(* Logix 5000 project; controller VET 1756-L62 rev 19.52; software revision 19.01; part 16 of 27 *)
(* tags used below, declared in another part *)
   _Eqp : Equipo[800];
   Batch : batch[10];
   dosificador : dosif_struct[20];
   Dosificar_MIC_02 : PHASE;
   Dosificar_MID_01 : PHASE;
   fecha_plc : DINT;
   hora_plc : DINT;
   SetDInt : DINT[500];
   TabBin : Bins_Setup;
   Timer : TIMER[500];
   vdf : VDFS[20];
(* Dosificar_MIC_02, continued *)

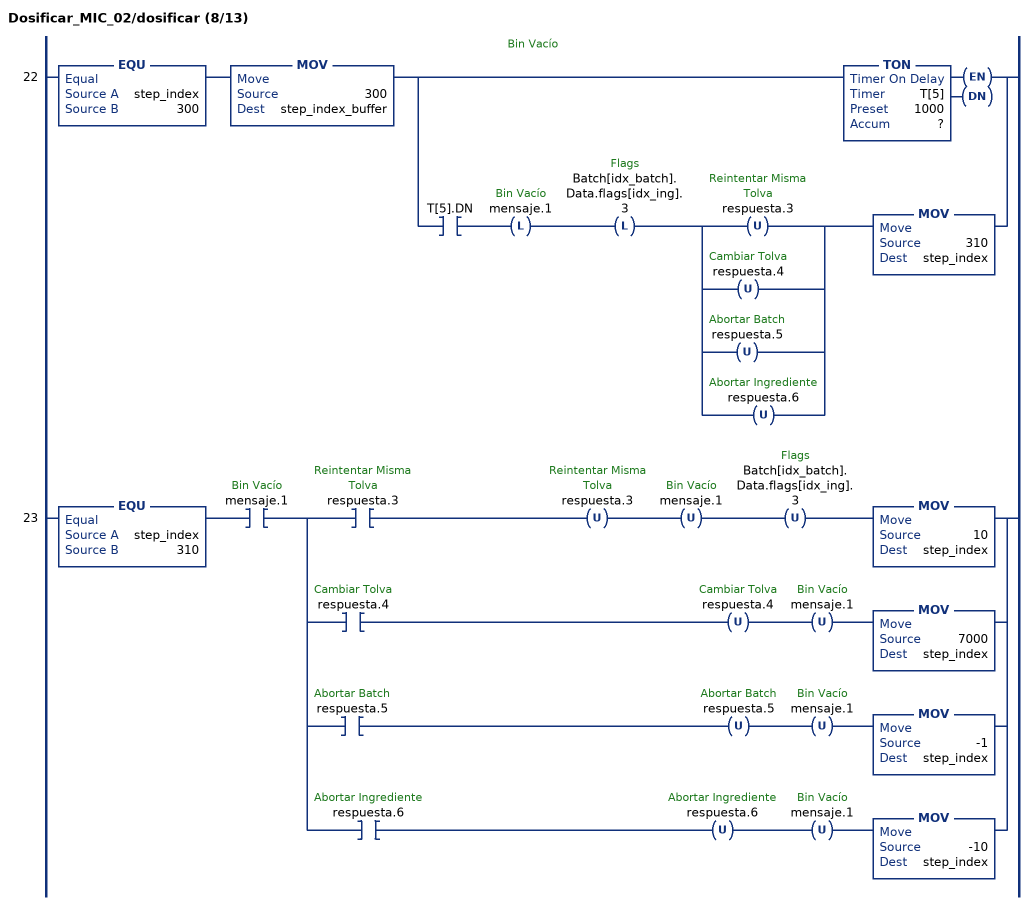
   // Bin Vacío
   22: EQU(step_index,300)MOV(300,step_index_buffer)[TON(T[5],?,?) ,XIC(T[5].DN) OTL(mensaje.1) OTL(Batch[idx_batch].Data.flags[idx_ing].3) [OTU(respuesta.3) ,OTU(respuesta.4) ,OTU(respuesta.5) ,OTU(respuesta.6) ] MOV(310,step_index) ];
   23: EQU(step_index,310)XIC(mensaje.1)[XIC(respuesta.3) OTU(respuesta.3) OTU(mensaje.1) OTU(Batch[idx_batch].Data.flags[idx_ing].3) MOV(10,step_index) ,XIC(respuesta.4) OTU(respuesta.4) OTU(mensaje.1) MOV(7000,step_index) ,XIC(respuesta.5) OTU(respuesta.5) OTU(mensaje.1) MOV(-1,step_index) ,XIC(respuesta.6) OTU(respuesta.6) OTU(mensaje.1) MOV(-10,step_index) ];
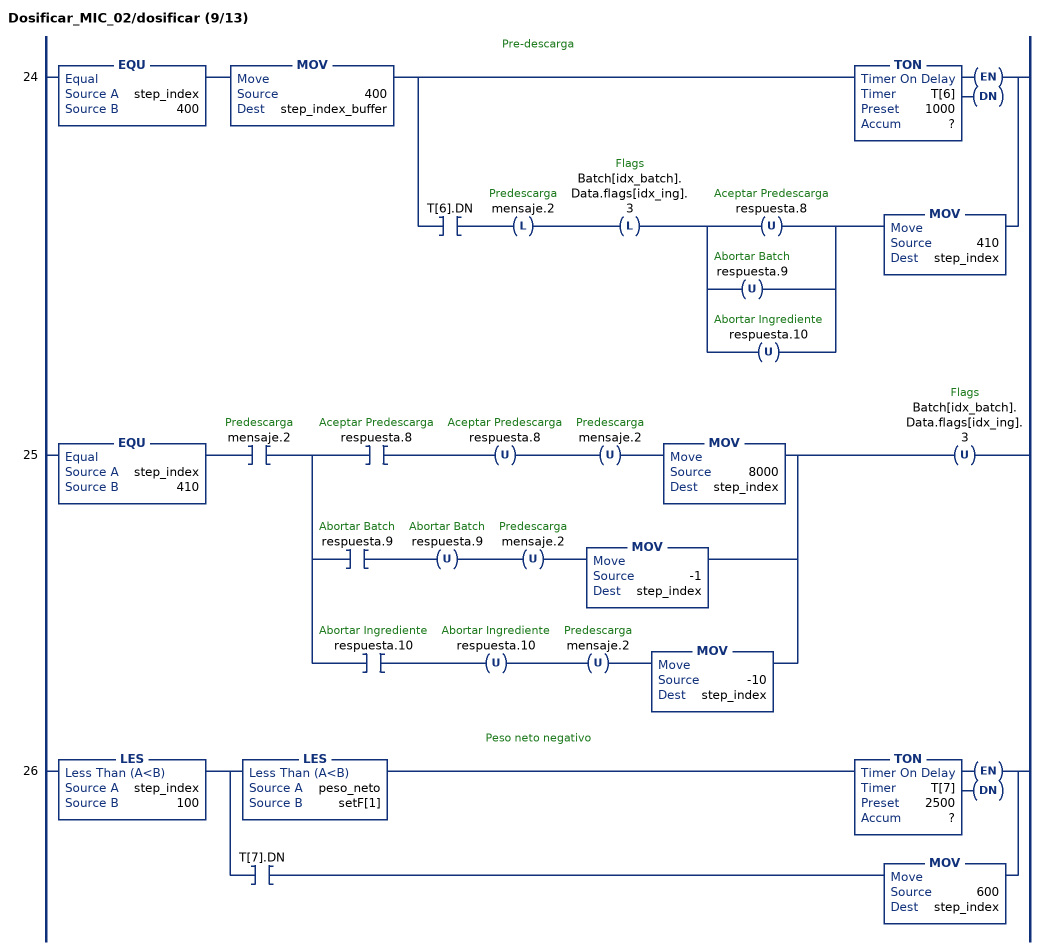
   // Pre-descarga
   24: EQU(step_index,400)MOV(400,step_index_buffer)[TON(T[6],?,?) ,XIC(T[6].DN) OTL(mensaje.2) OTL(Batch[idx_batch].Data.flags[idx_ing].3) [OTU(respuesta.8) ,OTU(respuesta.9) ,OTU(respuesta.10) ] MOV(410,step_index) ];
   25: EQU(step_index,410)XIC(mensaje.2)[XIC(respuesta.8) OTU(respuesta.8) OTU(mensaje.2) MOV(8000,step_index) ,XIC(respuesta.9) OTU(respuesta.9) OTU(mensaje.2) MOV(-1,step_index) ,XIC(respuesta.10) OTU(respuesta.10) OTU(mensaje.2) MOV(-10,step_index) ]OTU(Batch[idx_batch].Data.flags[idx_ing].3);
   // Peso neto negativo
   26: LES(step_index,100)[LES(peso_neto,setF[1]) TON(T[7],?,?) ,XIC(T[7].DN) MOV(600,step_index) ];
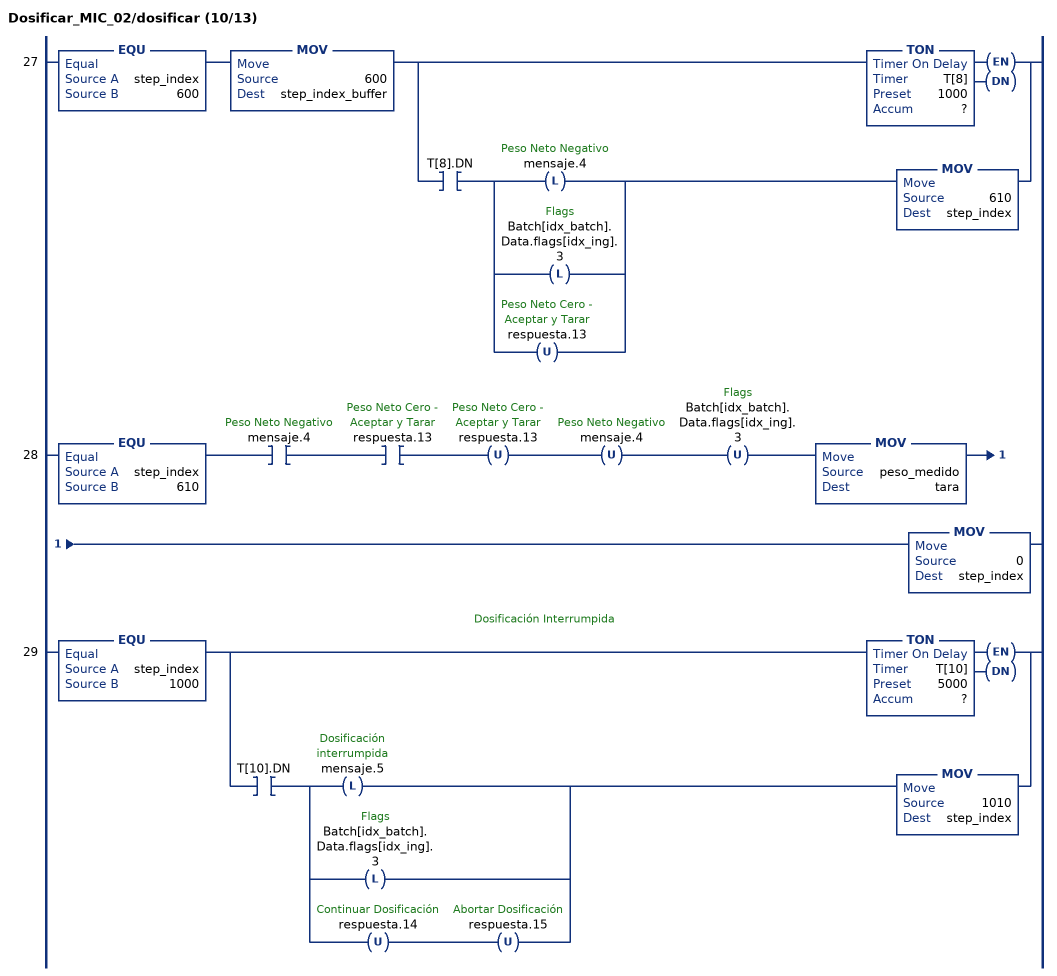
   27: EQU(step_index,600)MOV(600,step_index_buffer)[TON(T[8],?,?) ,XIC(T[8].DN) [OTL(mensaje.4) ,OTL(Batch[idx_batch].Data.flags[idx_ing].3) ,OTU(respuesta.13) ] MOV(610,step_index) ];
   28: EQU(step_index,610)XIC(mensaje.4)XIC(respuesta.13)OTU(respuesta.13)OTU(mensaje.4)OTU(Batch[idx_batch].Data.flags[idx_ing].3)MOV(peso_medido,tara)MOV(0,step_index);
   // Dosificación Interrumpida
   29: EQU(step_index,1000)[TON(T[10],?,?) ,XIC(T[10].DN) [OTL(mensaje.5) ,OTL(Batch[idx_batch].Data.flags[idx_ing].3) ,OTU(respuesta.14) OTU(respuesta.15) ] MOV(1010,step_index) ];
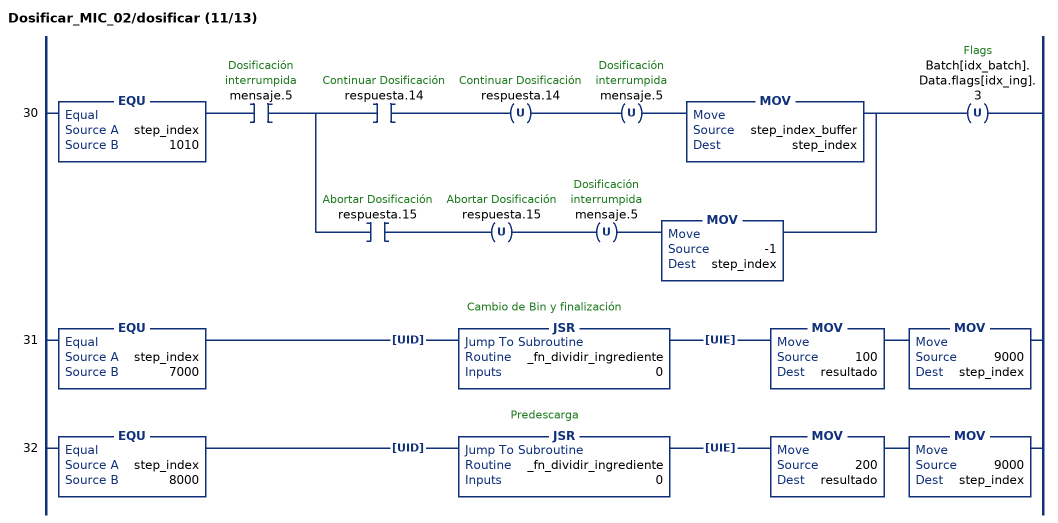
   30: EQU(step_index,1010)XIC(mensaje.5)[XIC(respuesta.14) OTU(respuesta.14) OTU(mensaje.5) MOV(step_index_buffer,step_index) ,XIC(respuesta.15) OTU(respuesta.15) OTU(mensaje.5) MOV(-1,step_index) ]OTU(Batch[idx_batch].Data.flags[idx_ing].3);
   // Cambio de Bin y finalización
   31: EQU(step_index,7000)UID()JSR(_fn_dividir_ingrediente,0)UIE()MOV(100,resultado)MOV(9000,step_index);
   // Predescarga
   32: EQU(step_index,8000)UID()JSR(_fn_dividir_ingrediente,0)UIE()MOV(200,resultado)MOV(9000,step_index);
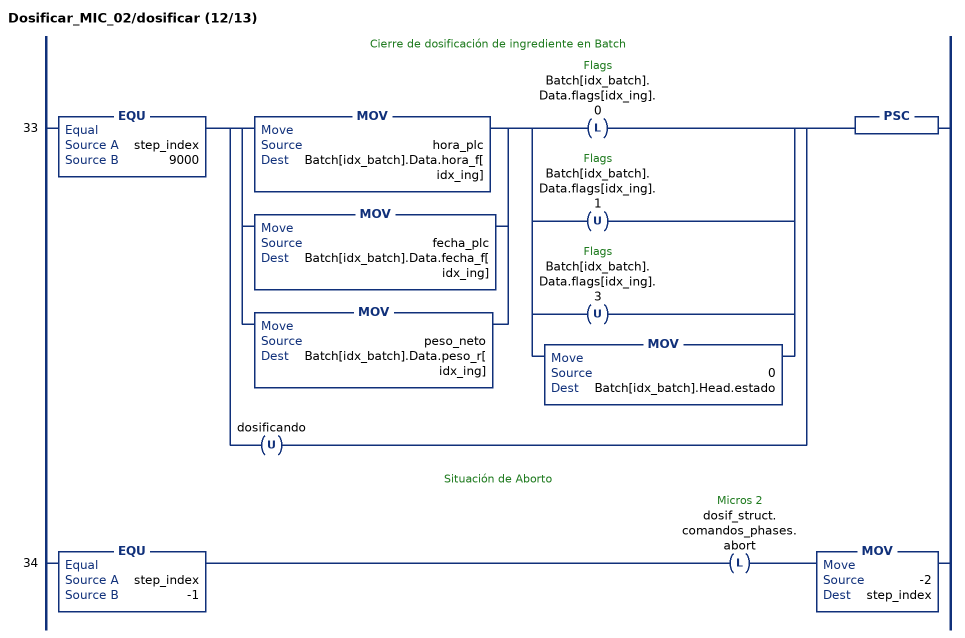
   // Cierre de dosificación de ingrediente en Batch
   33: EQU(step_index,9000)[[MOV(hora_plc,Batch[idx_batch].Data.hora_f[idx_ing]) ,MOV(fecha_plc,Batch[idx_batch].Data.fecha_f[idx_ing]) ,MOV(peso_neto,Batch[idx_batch].Data.peso_r[idx_ing]) ] [OTL(Batch[idx_batch].Data.flags[idx_ing].0) ,OTU(Batch[idx_batch].Data.flags[idx_ing].1) ,OTU(Batch[idx_batch].Data.flags[idx_ing].3) ,MOV(0,Batch[idx_batch].Head.estado) ] ,OTU(dosificando) ]PSC();
   // Situación de Aborto
   34: EQU(step_index,-1)OTL(dosif_struct.comandos_phases.abort)MOV(-2,step_index);
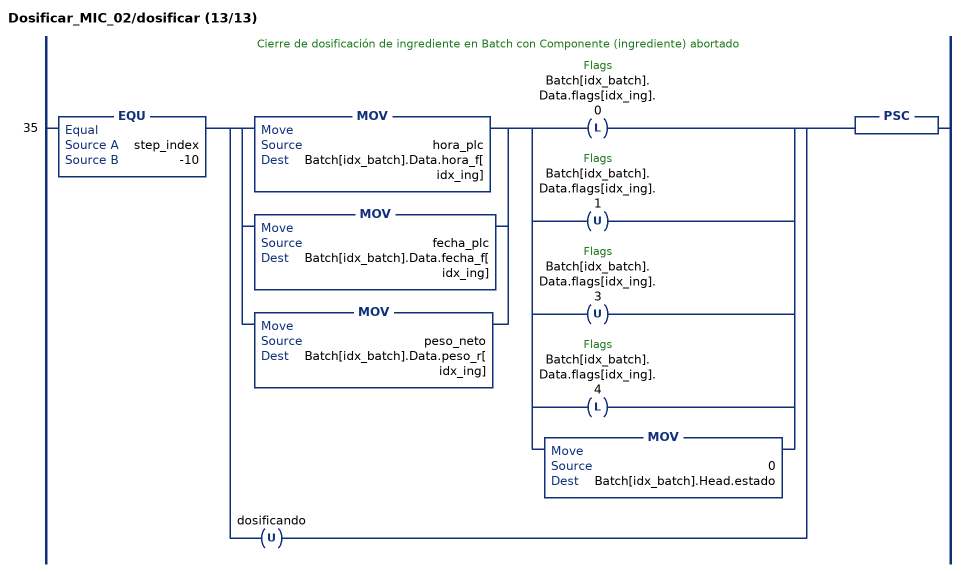
   // Cierre de dosificación de ingrediente en Batch con Componente (ingrediente) abortado
   35: EQU(step_index,-10)[[MOV(hora_plc,Batch[idx_batch].Data.hora_f[idx_ing]) ,MOV(fecha_plc,Batch[idx_batch].Data.fecha_f[idx_ing]) ,MOV(peso_neto,Batch[idx_batch].Data.peso_r[idx_ing]) ] [OTL(Batch[idx_batch].Data.flags[idx_ing].0) ,OTU(Batch[idx_batch].Data.flags[idx_ing].1) ,OTU(Batch[idx_batch].Data.flags[idx_ing].3) ,OTL(Batch[idx_batch].Data.flags[idx_ing].4) ,MOV(0,Batch[idx_batch].Head.estado) ] ,OTU(dosificando) ]PSC();
END_ROUTINE

ROUTINE Falla   (* ladder *)
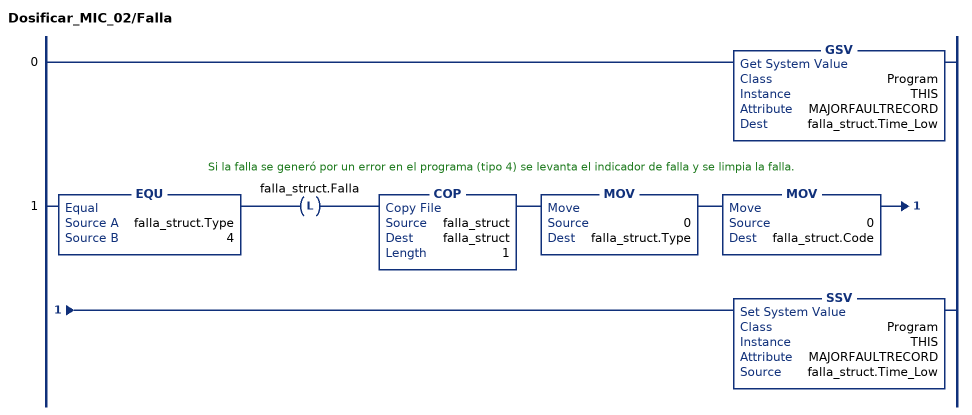
   0: GSV(Program,THIS,MAJORFAULTRECORD,falla_struct.Time_Low);
   // Si la falla se generó por un error en el programa (tipo 4) se levanta el indicador de falla y se limpia la falla.
   1: EQU(falla_struct.Type,4)OTL(falla_struct.Falla)COP(falla_struct,falla_struct,1)MOV(0,falla_struct.Type)MOV(0,falla_struct.Code)SSV(Program,THIS,MAJORFAULTRECORD,falla_struct.Time_Low);
END_ROUTINE

ROUTINE Holding   (* ladder *)
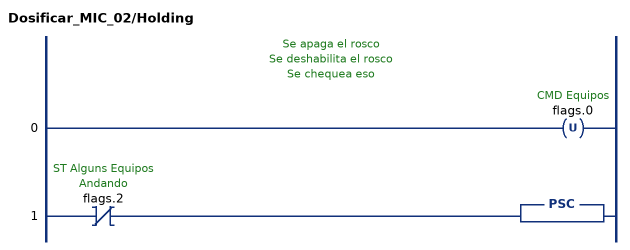
   // Se apaga el rosco
   // Se deshabilita el rosco
   // Se chequea eso
   0: OTU(flags.0);
   1: XIO(flags.2)PSC();
END_ROUTINE

ROUTINE preState   (* ladder *)
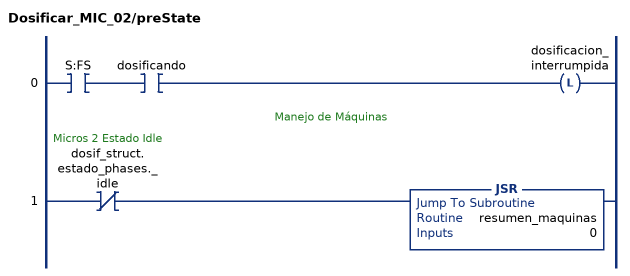
   0: XIC(S:FS)XIC(dosificando)OTL(dosificacion_interrumpida);
   // Manejo de Máquinas
   1: XIO(dosif_struct.estado_phases._idle)JSR(resumen_maquinas,0);
END_ROUTINE

ROUTINE Resetting   (* ladder *)
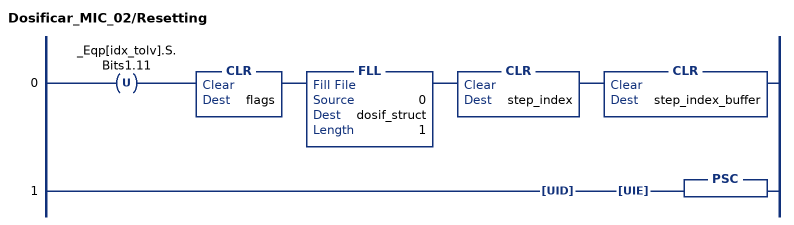
   0: OTU(_Eqp[idx_tolv].S.Bits1.11)CLR(flags)FLL(0,dosif_struct,1)CLR(step_index)CLR(step_index_buffer);
   1: UID()UIE()PSC();
END_ROUTINE

ROUTINE Restarting   (* ladder *)
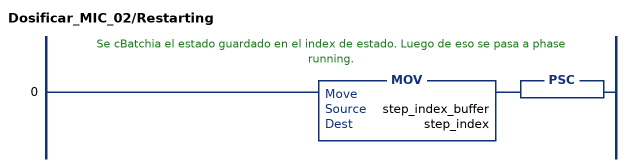
   // Se cBatchia el estado guardado en el index de estado. Luego de eso se pasa a phase running.
   0: MOV(step_index_buffer,step_index)PSC();
END_ROUTINE

ROUTINE resumen_maquinas   (* ladder *)
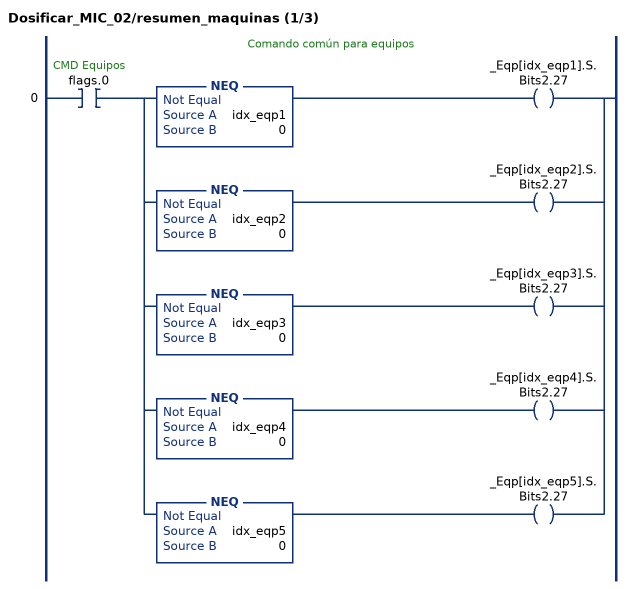
   // Comando común para equipos
   0: XIC(flags.0)[NEQ(idx_eqp1,0) OTE(_Eqp[idx_eqp1].S.Bits2.27) ,NEQ(idx_eqp2,0) OTE(_Eqp[idx_eqp2].S.Bits2.27) ,NEQ(idx_eqp3,0) OTE(_Eqp[idx_eqp3].S.Bits2.27) ,NEQ(idx_eqp4,0) OTE(_Eqp[idx_eqp4].S.Bits2.27) ,NEQ(idx_eqp5,0) OTE(_Eqp[idx_eqp5].S.Bits2.27) ];
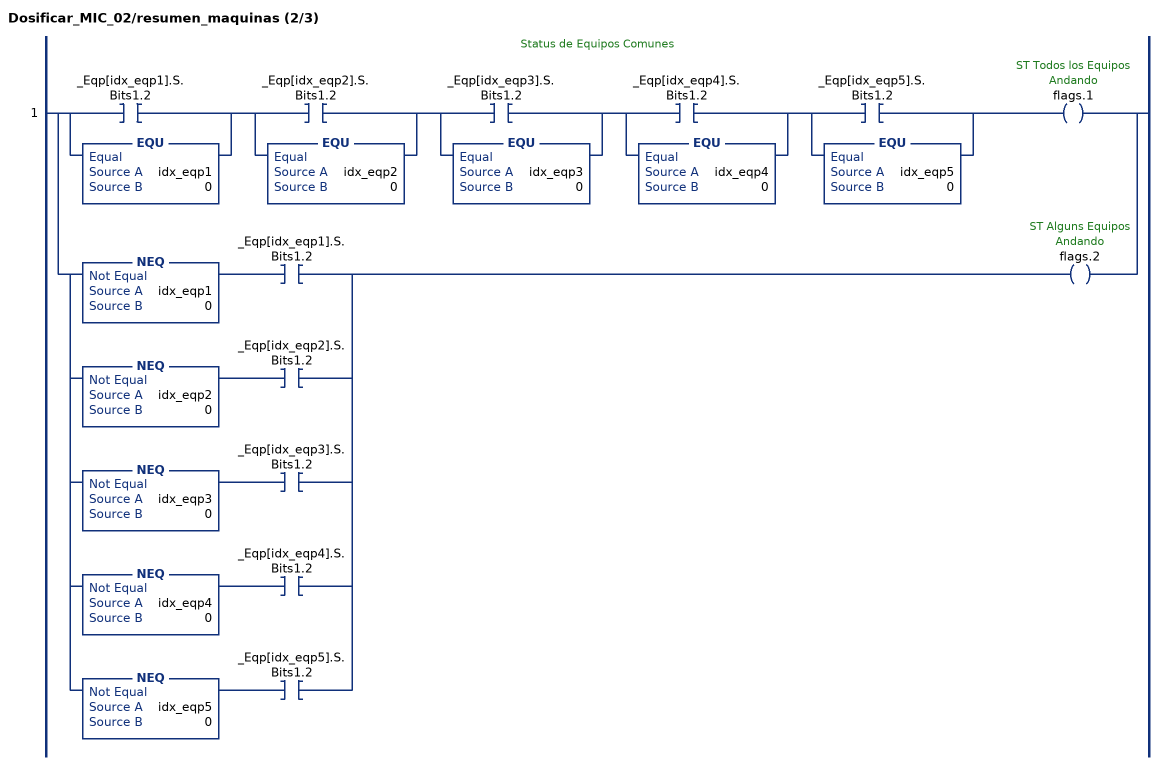
   // Status de Equipos Comunes
   1: [[XIC(_Eqp[idx_eqp1].S.Bits1.2) ,EQU(idx_eqp1,0) ] [XIC(_Eqp[idx_eqp2].S.Bits1.2) ,EQU(idx_eqp2,0) ] [XIC(_Eqp[idx_eqp3].S.Bits1.2) ,EQU(idx_eqp3,0) ] [XIC(_Eqp[idx_eqp4].S.Bits1.2) ,EQU(idx_eqp4,0) ] [XIC(_Eqp[idx_eqp5].S.Bits1.2) ,EQU(idx_eqp5,0) ] OTE(flags.1) ,[NEQ(idx_eqp1,0) XIC(_Eqp[idx_eqp1].S.Bits1.2) ,NEQ(idx_eqp2,0) XIC(_Eqp[idx_eqp2].S.Bits1.2) ,NEQ(idx_eqp3,0) XIC(_Eqp[idx_eqp3].S.Bits1.2) ,NEQ(idx_eqp4,0) XIC(_Eqp[idx_eqp4].S.Bits1.2) ,NEQ(idx_eqp5,0) XIC(_Eqp[idx_eqp5].S.Bits1.2) ] OTE(flags.2) ];
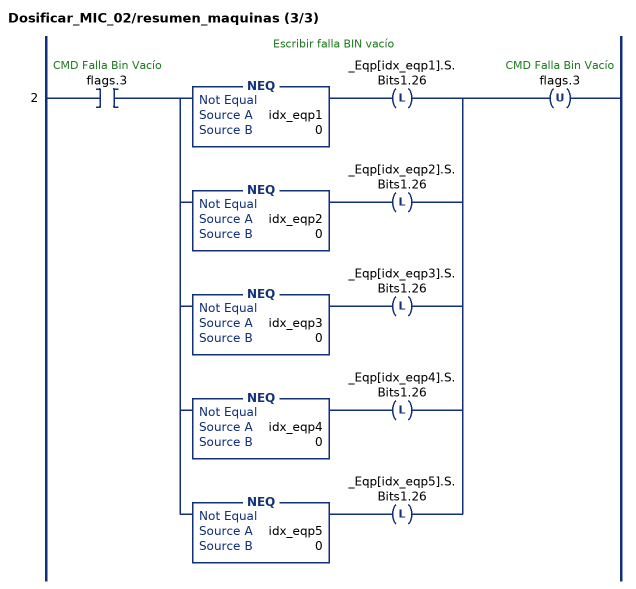
   // Escribir falla BIN vacío
   2: XIC(flags.3)[NEQ(idx_eqp1,0) OTL(_Eqp[idx_eqp1].S.Bits1.26) ,NEQ(idx_eqp2,0) OTL(_Eqp[idx_eqp2].S.Bits1.26) ,NEQ(idx_eqp3,0) OTL(_Eqp[idx_eqp3].S.Bits1.26) ,NEQ(idx_eqp4,0) OTL(_Eqp[idx_eqp4].S.Bits1.26) ,NEQ(idx_eqp5,0) OTL(_Eqp[idx_eqp5].S.Bits1.26) ]OTU(flags.3);
END_ROUTINE

ROUTINE Running   (* ladder *)
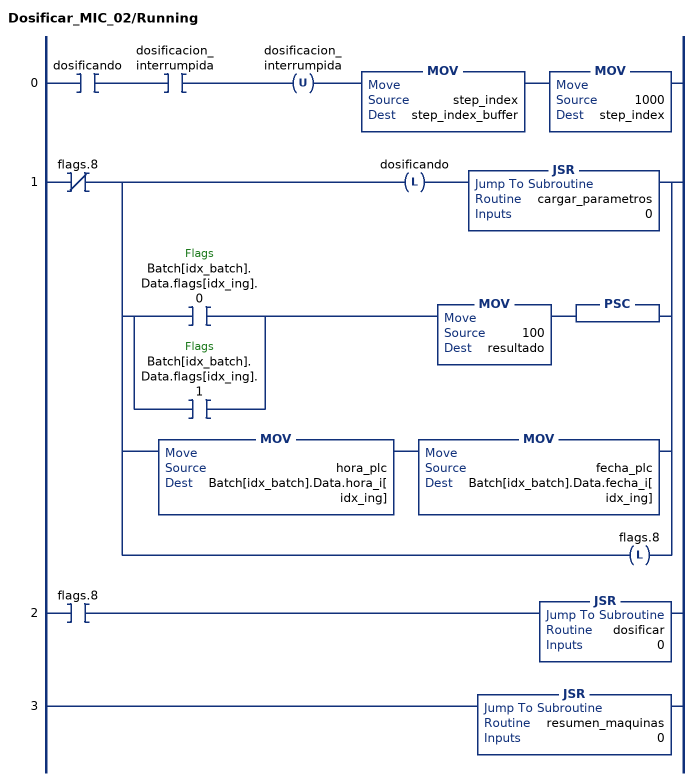
   0: XIC(dosificando)XIC(dosificacion_interrumpida)OTU(dosificacion_interrumpida)MOV(step_index,step_index_buffer)MOV(1000,step_index);
   1: XIO(flags.8)[OTL(dosificando) JSR(cargar_parametros,0) ,[[XIC(Batch[idx_batch].Data.flags[idx_ing].0) ,XIC(Batch[idx_batch].Data.flags[idx_ing].1) ] MOV(100,resultado) PSC() ,MOV(hora_plc,Batch[idx_batch].Data.hora_i[idx_ing]) MOV(fecha_plc,Batch[idx_batch].Data.fecha_i[idx_ing]) ] ,OTL(flags.8) ];
   2: XIC(flags.8)JSR(dosificar,0);
   3: JSR(resumen_maquinas,0);
END_ROUTINE
END_PROGRAM

PROGRAM Dosificar_MID_01   (* fault routine Falla *)
VAR
   _vel_exp : velocidad_exp := (x := 0.011880493, curvatura := 3.0, V_inicial := 70.0, V_final := 50.0, V_salida := 50.73287);
   bufferF : REAL[5] := ([0] := 90.78711, [1] := -0.7871094, [2] := 0.011880493);
        [2]   // Diferencia entre peso actual y objetivo
   debug : BOOL;
   dosif_extra_ingr : DINT := -1;   // Código del ingrediente que puede ser dosificado extra.
   dosif_struct : ALIAS FOR dosificador[1];
   dosificacion_interrumpida : BOOL;
   dosificando : BOOL;
   error_kg : REAL := 0.5;
   error_per : REAL := 4.5;
   falla_struct : falla_aux;
   flags : DINT;
        .1   // ST Todos los Equipos Andando
        .2   // ST Alguns Equipos Andando
        .3   // CMD Falla Bin Vacío
        .6   // Bit Precorte
        .7   // Aplicar Precorte
        .0   // CMD Equipos
   frq : ALIAS FOR dosif_struct.frq_terreno;
   frq_calculada : REAL := 50.0;
   frq_final : REAL := 50.0;
   frq_inicial : REAL := 70.0;
   hist_precorte : REAL[10] := ([0] := 1.0, [1] := 1.0, [2] := 1.0, [3] := 1.0, [4] := 1.0);
   i_fn : DINT;
   idx_batch : DINT := 3;
   idx_bin : DINT := 15;
   idx_dosif : DINT;   // Índice de dosificador usado
   idx_eqp1 : DINT := 53;
   idx_eqp2 : DINT;
   idx_eqp3 : DINT;
   idx_eqp4 : DINT;
   idx_eqp5 : DINT;
   idx_ing : DINT := 7;
   idx_tabbin : DINT := 1;
   idx_tolv : DINT := 34;   // Índice de Tolva
   limite_err_inf : REAL := 89.5;
   limite_err_sup : REAL := 90.5;
   mensaje : ALIAS FOR dosif_struct.msg;
        .1   // Bin Vacío
        .4   // Peso Neto Negativo
        .0   // Error de Pesaje
        .5   // Dosificación interrumpida
        .3   // Manual
        .2   // Predescarga
   peso_delta : REAL;
   peso_detencion : REAL := 89.09469;
   peso_intermedio : REAL := 54.000004;   // Peso límite para dosificación a frecuencia máxima
   peso_max : REAL := 700.0;
   peso_medido : ALIAS FOR dosif_struct.peso_terreno;
   peso_neto : REAL := 90.78711;
   peso_neto_aux : REAL;   // Peso Neto Guardado en caso de Vaciado y llenado de tolva
   peso_objetivo : REAL := 90.0;
   precorte : REAL := 1.102089;
   respuesta : ALIAS FOR dosif_struct.ans;
        .16   // Abortar Ingrediente
        .3   // Reintentar Misma Tolva
        .7   // Pasar a Manual
        .0   // Aceptar Error
        .14   // Continuar Dosificación
        .11   // Dosificación Completa
        .1   // Abortar Batch
        .2   // Abortar Ingrediente
        .12   // Habilitar Aceptar
        .8   // Aceptar Predescarga
        .10   // Abortar Ingrediente
        .5   // Abortar Batch
        .4   // Cambiar Tolva
        .6   // Abortar Ingrediente
        .15   // Abortar Dosificación
        .9   // Abortar Batch
        .13   // Peso Neto Cero - Aceptar y Tarar
   resultado : ALIAS FOR dosif_struct.resultado;
   return_fn : DINT;
   setD : DINT[5] := ([0] := 1, [1] := 44, [2] := 2, [3] := 1, [4] := 32);
        [1].3   // Aplicar Precorte
        [1].8   // Con VDF
        [4]   // Destino
        [1].2   // Predescarga
        [1].4   // Con Bloqueo de Tolva
        [1].5   // No respeta receta
        [2]   // Mezcladora izquierda
        [3]   // Mezcladora derecha
        [1].0   // Tipo LIW
        [0]   // Mínima variación de peso para detección de tolva vacía.
   setF : REAL[5] := ([0] := 1.0);
        [0]   // Límite para variación de peso
        [1]   // Límite para peso negativo
   step_index : DINT;
   step_index_buffer : DINT;
   T : TIMER[15] := ([0].PRE := 1000, [0].ACC := 80, [0].EN := 1, [0].TT := 1, [1].PRE := 30000, [2].PRE := 3000, [3].PRE := 10000, [4].PRE := 1000, [5].PRE := 1000, [6].PRE := 1000, [7].PRE := 2500, [8].PRE := 1000, [9].PRE := 1000, [10].PRE := 5000);
   t_espera : DINT := 3000;
   t_pulso : DINT := 10000;
   tara : REAL := 360.85922;
END_VAR

ROUTINE _fn_dividir_ingrediente   (* ladder *)
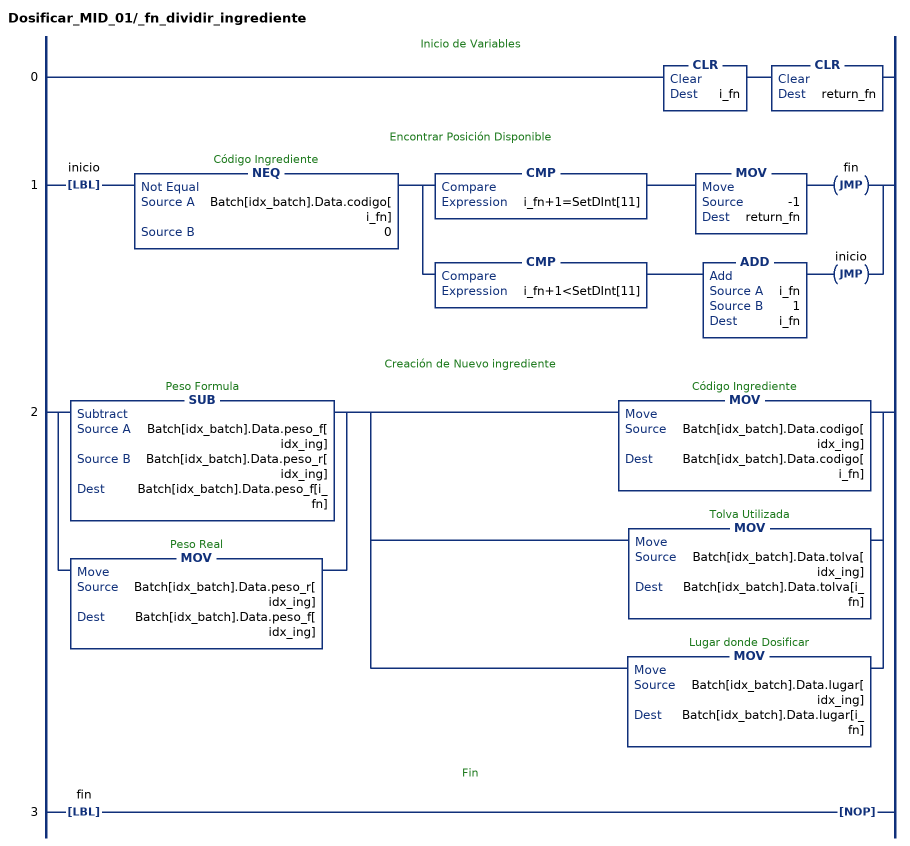
   // Inicio de Variables
   0: CLR(i_fn)CLR(return_fn);
   // Encontrar Posición Disponible
   1: LBL(inicio)NEQ(Batch[idx_batch].Data.codigo[i_fn],0)[CMP(i_fn+1=SetDInt[11]) MOV(-1,return_fn) JMP(fin) ,CMP(i_fn+1<SetDInt[11]) ADD(i_fn,1,i_fn) JMP(inicio) ];
   // Creación de Nuevo ingrediente
   2: [SUB(Batch[idx_batch].Data.peso_f[idx_ing],Batch[idx_batch].Data.peso_r[idx_ing],Batch[idx_batch].Data.peso_f[i_fn]) ,MOV(Batch[idx_batch].Data.peso_r[idx_ing],Batch[idx_batch].Data.peso_f[idx_ing]) ][MOV(Batch[idx_batch].Data.codigo[idx_ing],Batch[idx_batch].Data.codigo[i_fn]) ,MOV(Batch[idx_batch].Data.tolva[idx_ing],Batch[idx_batch].Data.tolva[i_fn]) ,MOV(Batch[idx_batch].Data.lugar[idx_ing],Batch[idx_batch].Data.lugar[i_fn]) ];
   // Fin
   3: LBL(fin)NOP();
END_ROUTINE

ROUTINE Aborting   (* ladder *)
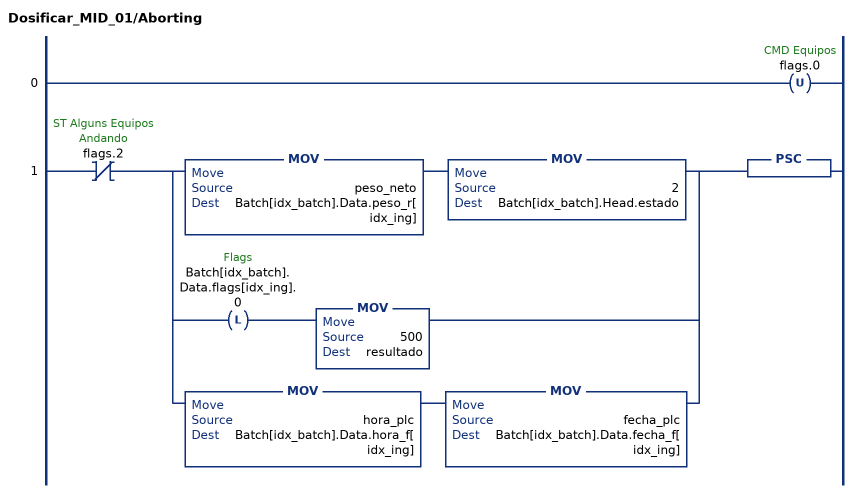
   0: OTU(flags.0);
   1: XIO(flags.2)[MOV(peso_neto,Batch[idx_batch].Data.peso_r[idx_ing]) MOV(2,Batch[idx_batch].Head.estado) ,OTL(Batch[idx_batch].Data.flags[idx_ing].0) MOV(500,resultado) ,MOV(hora_plc,Batch[idx_batch].Data.hora_f[idx_ing]) MOV(fecha_plc,Batch[idx_batch].Data.fecha_f[idx_ing]) ]PSC();
END_ROUTINE

ROUTINE calculo_frecuencia   (* ladder *)
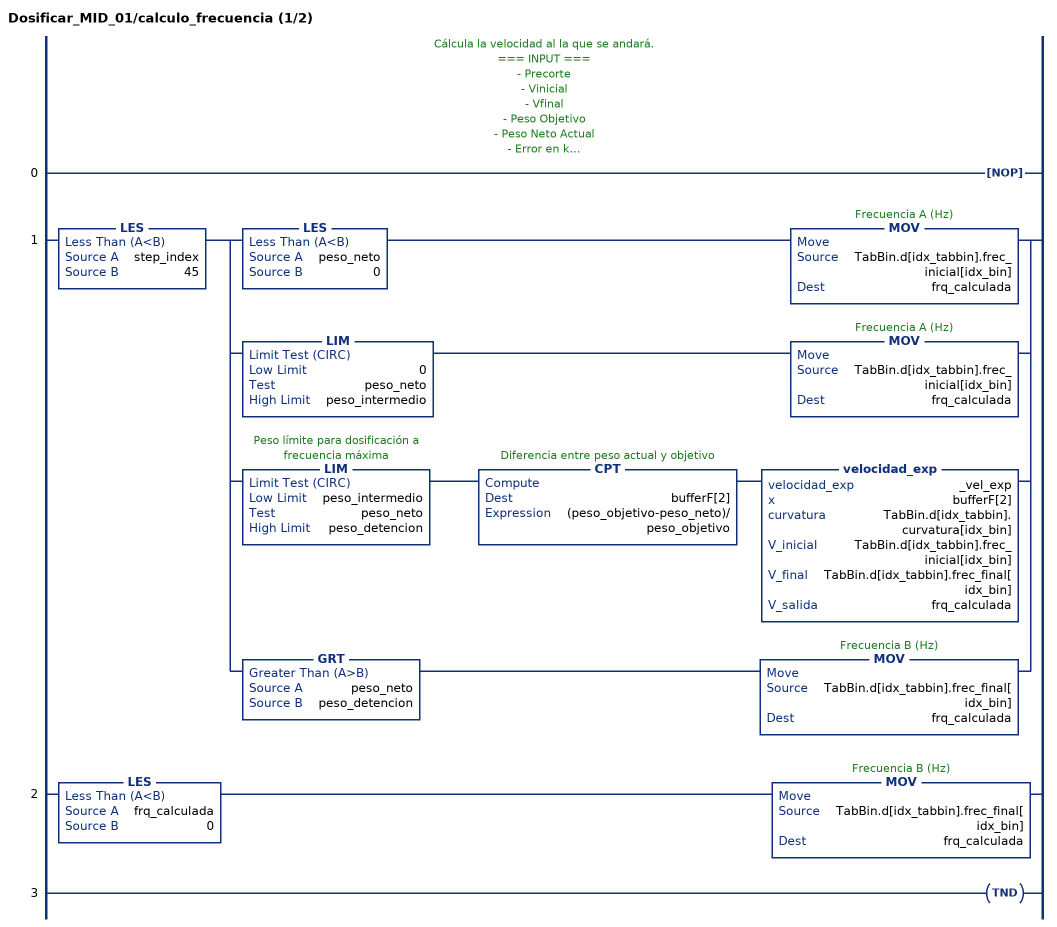
   // Cálcula la velocidad al la que se andará.
   // === INPUT ===
   // - Precorte
   // - Vinicial
   // - Vfinal
   // - Peso Objetivo
   // - Peso Neto Actual
   // - Error en kg
   // === OUTPUT ===
   // - Vactual
   0: NOP();
   1: LES(step_index,45)[LES(peso_neto,0) MOV(TabBin.d[idx_tabbin].frec_inicial[idx_bin],frq_calculada) ,LIM(0,peso_neto,peso_intermedio) MOV(TabBin.d[idx_tabbin].frec_inicial[idx_bin],frq_calculada) ,LIM(peso_intermedio,peso_neto,peso_detencion) CPT(bufferF[2],(peso_objetivo-peso_neto)/peso_objetivo) velocidad_exp(_vel_exp,bufferF[2],TabBin.d[idx_tabbin].curvatura[idx_bin],TabBin.d[idx_tabbin].frec_inicial[idx_bin],TabBin.d[idx_tabbin].frec_final[idx_bin],frq_calculada) ,GRT(peso_neto,peso_detencion) MOV(TabBin.d[idx_tabbin].frec_final[idx_bin],frq_calculada) ];
   2: LES(frq_calculada,0)MOV(TabBin.d[idx_tabbin].frec_final[idx_bin],frq_calculada);
   3: TND();
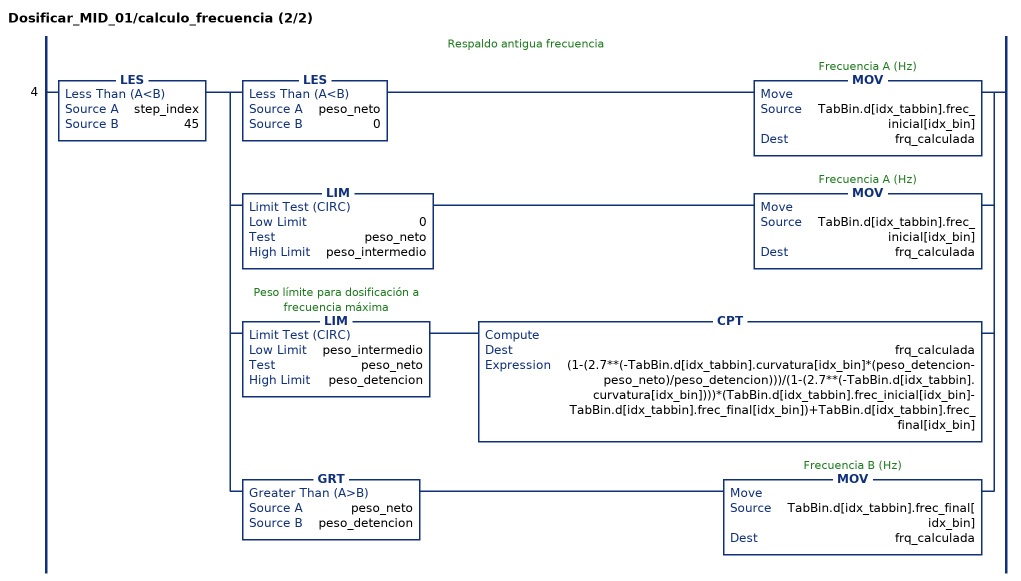
   // Respaldo antigua frecuencia
   4: LES(step_index,45)[LES(peso_neto,0) MOV(TabBin.d[idx_tabbin].frec_inicial[idx_bin],frq_calculada) ,LIM(0,peso_neto,peso_intermedio) MOV(TabBin.d[idx_tabbin].frec_inicial[idx_bin],frq_calculada) ,LIM(peso_intermedio,peso_neto,peso_detencion) CPT(frq_calculada,(1-(2.7**(-TabBin.d[idx_tabbin].curvatura[idx_bin]*(peso_detencion-peso_neto)/peso_detencion)))/(1-(2.7**(-TabBin.d[idx_tabbin].curvatura[idx_bin])))*(TabBin.d[idx_tabbin].frec_inicial[idx_bin]-TabBin.d[idx_tabbin].frec_final[idx_bin])+TabBin.d[idx_tabbin].frec_final[idx_bin]) ,GRT(peso_neto,peso_detencion) MOV(TabBin.d[idx_tabbin].frec_final[idx_bin],frq_calculada) ];
END_ROUTINE
